# EPICS StreamDevice protocol: siteApps/KoBRA_MAG-1-0/proto/danfysikMps8700_scpi.proto
#
#

#8700 IP(192.168.131.20), PORT(13000)

#OutTerminator = CR LF;
#InTerminator  = CR LF;
Terminator = CR LF;
ReplyTimeout  = 1000;
ReadTimeout   = 100;
WriteTimeout  = 100;
LockTimeout   = 5000;

setcmd		{ out "%{LOC|REM}";							}
getcmd		{ out "CMD";			in "%{LOC|REM} ";	}

power		{ out "OUTP:REL			%{OFF|ON}";			}
rdpower		{ out "OUTP:REL?";		in "%d";			}

getcurr		{ out "MEAS:CURR?";		in "%f";			}
getvolt		{ out "MEAS:VOLT?";		in "%f";			}

setcurr		{ out "CURR %03d";							}
setcurrRB	{ out "CURR?";			in "%f"				}

status	    { out "STAT?";			in "%d";			}
reg1	    { out "STAT:OPER:REG1?";in "%d";			}
reg2	    { out "STAT:OPER:REG2?";in "%d";			}
reg3	    { out "STAT:OPER:REG3?";in "%d";			}
